PROGRAM PRG_DE_TESTES
VAR
	Lavagem:Lavagem;
	Calibracao: Calibracao_V02;
	FB_DBRead_0: FB_DBRead;
	grupo:STRING;
	hora:TIME;
	data:DATE;
	nome:STRING;
	mensagem:LREAL;
	EventLog:DINT;
	FB_DBConnectionAdd_0: FB_DBConnectionAdd;
	FB_DBCyclicRdWrt_0: FB_DBCyclicRdWrt;
	FB_DBConnectionAdd_1: FB_DBConnectionAdd;
	TesteAlarmes : ARRAY [1..3 ] OF GeraAlarme;
	AcionaEvento: BOOL;
	Confirma: BOOL;
	MediaMovel_0: MediaMovel;
	TON_teste: TON;
	SDO_READ_0: SDO_READ;
	FB_EcCoESdoRead_0: FB_EcCoESdoRead;
	SDO_READ_1: SDO_READ;
	Calibracao_V03_0: Calibracao_V03;
	DiagInfo:STRING;
	TesteApex:INT;
	FB_IPCDiag_ReadParameter_0: FB_IPCDiag_ReadParameter;
	fbRegister: FB_IPCDiag_Register;
END_VAR
VAR // added by the converter: edge detectors and wires of the graphical bodies
    _w1, _w2 : BOOL;
END_VAR

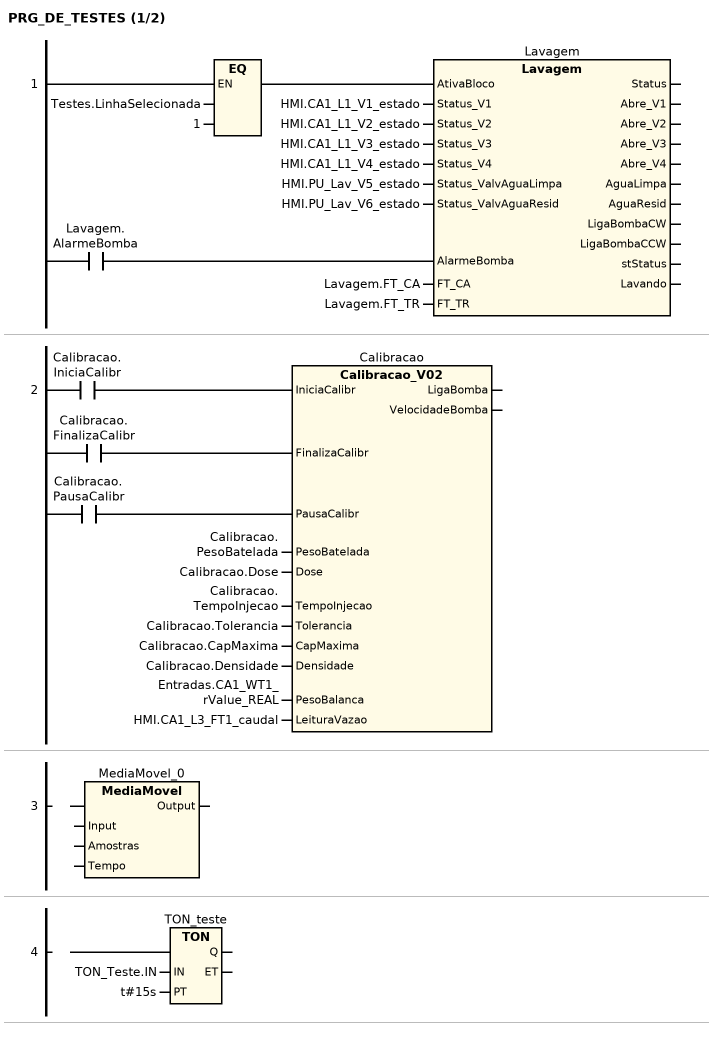
// NETWORK 1
Lavagem(
    AtivaBloco := Testes.LinhaSelecionada = 1,
    Status_V1 := HMI.CA1_L1_V1_estado,
    Status_V2 := HMI.CA1_L1_V2_estado,
    Status_V3 := HMI.CA1_L1_V3_estado,
    Status_V4 := HMI.CA1_L1_V4_estado,
    Status_ValvAguaLimpa := HMI.PU_Lav_V5_estado,
    Status_ValvAguaResid := HMI.PU_Lav_V6_estado,
    AlarmeBomba := Lavagem.AlarmeBomba,
    FT_CA := Lavagem.FT_CA,
    FT_TR := Lavagem.FT_TR);

// NETWORK 2
Calibracao(
    IniciaCalibr := Calibracao.IniciaCalibr,
    FinalizaCalibr := Calibracao.FinalizaCalibr,
    PausaCalibr := Calibracao.PausaCalibr,
    PesoBatelada := Calibracao.PesoBatelada,
    Dose := Calibracao.Dose,
    TempoInjecao := Calibracao.TempoInjecao,
    Tolerancia := Calibracao.Tolerancia,
    CapMaxima := Calibracao.CapMaxima,
    Densidade := Calibracao.Densidade,
    PesoBalanca := Entradas.CA1_WT1_rValue_REAL,
    LeituraVazao := HMI.CA1_L3_FT1_caudal); // Calibracao_V02

// NETWORK 3
MediaMovel_0(); // MediaMovel

// NETWORK 4
TON_teste(IN := TON_Teste.IN, PT := t#15s); // TON

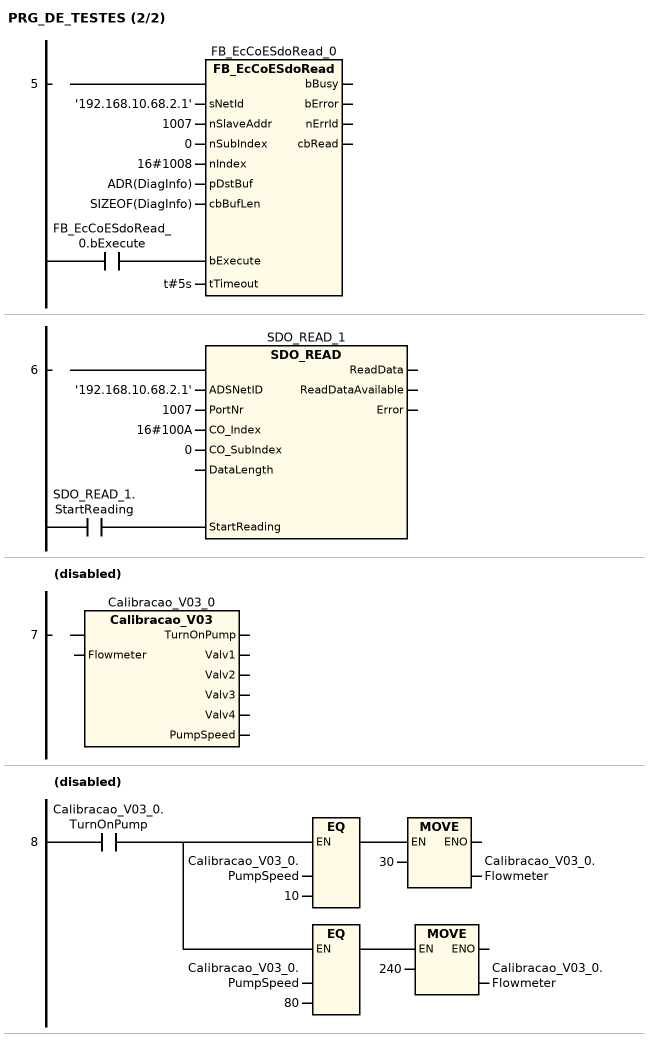
// NETWORK 5
FB_EcCoESdoRead_0(
    sNetId := '192.168.10.68.2.1',
    nSlaveAddr := 1007,
    nSubIndex := 0,
    nIndex := 16#1008,
    pDstBuf := ADR(DiagInfo),
    cbBufLen := SIZEOF(DiagInfo),
    bExecute := FB_EcCoESdoRead_0.bExecute,
    tTimeout := t#5s); // FB_EcCoESdoRead

// NETWORK 6
SDO_READ_1(
    ADSNetID := '192.168.10.68.2.1',
    PortNr := 1007,
    CO_Index := 16#100A,
    CO_SubIndex := 0,
    StartReading := SDO_READ_1.StartReading); // SDO_READ

// NETWORK 7 (disabled)
// Calibracao_V03_0(); // Calibracao_V03

// NETWORK 8 (disabled)
// _w1 := Calibracao_V03_0.TurnOnPump AND Calibracao_V03_0.PumpSpeed = 10;
// IF _w1 THEN Calibracao_V03_0.Flowmeter := 30; END_IF
// _w2 := Calibracao_V03_0.TurnOnPump AND Calibracao_V03_0.PumpSpeed = 80;
// IF _w2 THEN Calibracao_V03_0.Flowmeter := 240; END_IF

END_PROGRAM

(* stored: Version 1.1.0.1, ProductVersion 3.1.4024.14
   POU PRG_DE_TESTES: Id {845a1b45-45c9-4d8f-93ca-a1b1e36e4802}, SpecialFunc None *)
